Universal Robots PolyScope program: move down.urp

Program move_down (installation=assignment directory=/home/mtrn4230/ursim-5.10.0.106288/programs createdIn=5.10.0.106288 lastSavedIn=5.10.0.106288 robotSerialNumber=20195599999)
Calibrated DH parameters: a=[0, -0.425, -0.3922, 0, 0, 0]; d=[0.1625, 0, 0, 0.1333, 0.0997, 0.0996]; alpha=[1.570796, 0, 0, 1.570796, -1.570796, 0]; deltaTheta=[0, 0, 0, 0, 0, 0]
Robot Program (runOnlyOnce=false)
  curr_pos := pose_trans(pose_sub(get_actual_tcp_pose(), letter_start), p[0,0,-1/100,0,0,0])
  MoveL speed 250 mm/s, acceleration 1200 mm/s^2 (useActiveTCP=true) feature=letter_start
    Waypoint Waypoint (Variable): variable=curr_pos
